// TIA Portal V15.1 export
// export: Created 2024-05-17T05:38:33.441184Z, ExportSetting WithDefaults, DisplayName Totally Integrated Automation Portal, DisplayVersion V15.1 Update 5, DisplayName TIA Portal Openness, DisplayVersion V15.1 Update 5, DisplayName SINAMICS Startdrive Advanced, DisplayVersion V15.1, DisplayName G130, G150, S120, S150, SINAMICS MV, S210, DisplayVersion V15.1, DisplayName G110M, G120, G120C, G120D, G120P, DisplayVersion V15.1, DisplayName STEP 7 Professional, DisplayVersion V15.1 Update 5, DisplayName STEP 7 Safety, DisplayVersion V15.1, DisplayName WinCC Professional, DisplayVersion V15.1 Update 5, DisplayName SIMATIC Visualization Architect, DisplayVersion V15.1
FUNCTION_BLOCK "LProcMasterSlave"   // FB1706, FBD
TITLE = LProcMasterSlave
{ S7_Optimized_Access := 'FALSE' }
AUTHOR : VCC
FAMILY : Control
NAME : MSCtrl
VERSION : 0.1
// ================================================================================
// Master-Slave Controller:
// The temperature is controlled by the Master continuous controller CONT_C and 
// puts out a setpoint value 0-100% to the slave controller CONT_S.
// ================================================================================
// stored: AutoNumber false, IsIECCheckEnabled false, SetENOAutomatically False, UDAEnableTagReadback false
   VAR_INPUT
      I_CYCLE { ExternalAccessible := 'False'; ExternalVisible := 'False'; ExternalWritable := 'False'} : Time;   // Sample time
      I_M_SP_Manual { ExternalAccessible := 'False'; ExternalVisible := 'False'; ExternalWritable := 'False'} : Real;   // Master: Setpoint Manual
      I_M_SP_Auto { ExternalAccessible := 'False'; ExternalVisible := 'False'; ExternalWritable := 'False'} : Real;   // Master: Setpoint for controller
      I_M_PV { ExternalAccessible := 'False'; ExternalVisible := 'False'; ExternalWritable := 'False'} : Real;   // Master: Process value
      I_M_GAIN { ExternalAccessible := 'False'; ExternalVisible := 'False'; ExternalWritable := 'False'} : Real;   // Master: Proportional Gain
      I_M_TI { ExternalAccessible := 'False'; ExternalVisible := 'False'; ExternalWritable := 'False'} : Time;   // Master: Reset time
      I_M_TD { ExternalAccessible := 'False'; ExternalVisible := 'False'; ExternalWritable := 'False'} : Time;   // Master: Derivative time
      I_M_TM_LAG { ExternalAccessible := 'False'; ExternalVisible := 'False'; ExternalWritable := 'False'} : Time;   // Master: Time lag of the derivative action
      I_M_DEADB_W { ExternalAccessible := 'False'; ExternalVisible := 'False'; ExternalWritable := 'False'} : Real;   // Master: Deadband width
      I_M_LMN_HLM { ExternalAccessible := 'False'; ExternalVisible := 'False'; ExternalWritable := 'False'} : Real := 100.0;   // Master: Manipulated value high limit
      I_M_LMN_LLM { ExternalAccessible := 'False'; ExternalVisible := 'False'; ExternalWritable := 'False'} : Real;   // Master: Manipulated value low limit
      I_M_ER_MAX { ExternalAccessible := 'False'; ExternalVisible := 'False'; ExternalWritable := 'False'} : Real := 10.0;   // Master: Maximum deviation for error signal
      I_S_PV { ExternalAccessible := 'False'; ExternalVisible := 'False'; ExternalWritable := 'False'} : Real;   // Slave: Process value
      I_S_GAIN { ExternalAccessible := 'False'; ExternalVisible := 'False'; ExternalWritable := 'False'} : Real;   // Slave: Proportional Gain
      I_S_TI { ExternalAccessible := 'False'; ExternalVisible := 'False'; ExternalWritable := 'False'} : Time;   // Slave: Reset time
      I_S_DEADB_W { ExternalAccessible := 'False'; ExternalVisible := 'False'; ExternalWritable := 'False'} : Real;   // Slave: Deadband width
      I_S_ER_MAX { ExternalAccessible := 'False'; ExternalVisible := 'False'; ExternalWritable := 'False'} : Real := 10.0;   // Slave: Maximum deviation for error signal
      I_S_PULSE_TM { ExternalAccessible := 'False'; ExternalVisible := 'False'; ExternalWritable := 'False'} : Time;   // Slave: Minimum Pulse Time
      I_S_BREAK_TM { ExternalAccessible := 'False'; ExternalVisible := 'False'; ExternalWritable := 'False'} : Time;   // Slave: Minimum Break Time
      I_S_MTR_TM { ExternalAccessible := 'False'; ExternalVisible := 'False'; ExternalWritable := 'False'} : Time;   // Slave: Motor manipulated value
      I_COM_RST { ExternalAccessible := 'False'; ExternalVisible := 'False'; ExternalWritable := 'False'} : Bool;   // Initialising reset of controller
      I_M_MAN_ON { ExternalAccessible := 'False'; ExternalVisible := 'False'; ExternalWritable := 'False'} : Bool;   // Master: Manual value on
      I_M_P_SEL { ExternalAccessible := 'False'; ExternalVisible := 'False'; ExternalWritable := 'False'} : Bool;   // Master: P selected
      I_M_I_SEL { ExternalAccessible := 'False'; ExternalVisible := 'False'; ExternalWritable := 'False'} : Bool;   // Master: I selected
      I_M_D_SEL { ExternalAccessible := 'False'; ExternalVisible := 'False'; ExternalWritable := 'False'} : Bool;   // Master: D selected
      I_S_LMNR_HS { ExternalAccessible := 'False'; ExternalVisible := 'False'; ExternalWritable := 'False'} : Bool;   // Slave: Digital feedback MAX, I/O
      I_S_LMNR_LS { ExternalAccessible := 'False'; ExternalVisible := 'False'; ExternalWritable := 'False'} : Bool;   // Slave: Digital feedback MIN, I/O
      I_S_LMNUP { ExternalAccessible := 'False'; ExternalVisible := 'False'; ExternalWritable := 'False'} : Bool;   // Slave: Manipulated signal up
      I_S_LMNDN { ExternalAccessible := 'False'; ExternalVisible := 'False'; ExternalWritable := 'False'} : Bool;   // Slave: Manipulated signal down
   END_VAR
   VAR_OUTPUT
      O_M_ER { ExternalAccessible := 'False'; ExternalVisible := 'False'; ExternalWritable := 'False'} : Real;   // Deviation Master Controller
      O_SP { ExternalAccessible := 'False'; ExternalVisible := 'False'; ExternalWritable := 'False'} : Real;   // Setpoint used in controller
      O_QLMNUP { ExternalAccessible := 'False'; ExternalVisible := 'False'; ExternalWritable := 'False'} : Bool;   // Output Open
      O_QLMNDN { ExternalAccessible := 'False'; ExternalVisible := 'False'; ExternalWritable := 'False'} : Bool;   // Output Close
      O_M_ER_Alarm { ExternalAccessible := 'False'; ExternalVisible := 'False'; ExternalWritable := 'False'} : Bool;   // Master alarm for deviation
      O_S_ER_Alarm { ExternalAccessible := 'False'; ExternalVisible := 'False'; ExternalWritable := 'False'} : Bool;   // Slave alarm for deviation
   END_VAR
   VAR DB_SPECIFIC
      M_ManValue { ExternalAccessible := 'False'; ExternalVisible := 'False'; ExternalWritable := 'False'} : Real;   // Master: Manual value
      M_LMN { ExternalAccessible := 'False'; ExternalVisible := 'False'; ExternalWritable := 'False'} : Real;   // Master: Manipulated value from controller
      M_PV { ExternalAccessible := 'False'; ExternalVisible := 'False'; ExternalWritable := 'False'} : Real;   // Master: Process variable from controller
      M_ER { ExternalAccessible := 'False'; ExternalVisible := 'False'; ExternalWritable := 'False'} : Real;   // Master: Error signal from controller
      M_ER_ABS { ExternalAccessible := 'False'; ExternalVisible := 'False'; ExternalWritable := 'False'} : Real;   // Master: Absolute error from controller
      S_PV { ExternalAccessible := 'False'; ExternalVisible := 'False'; ExternalWritable := 'False'} : Real;   // Slave: Process variable from controller
      S_ER { ExternalAccessible := 'False'; ExternalVisible := 'False'; ExternalWritable := 'False'} : Real;   // Slave: Error signal from controller
      S_ER_ABS { ExternalAccessible := 'False'; ExternalVisible := 'False'; ExternalWritable := 'False'} : Real;   // Slave: Absolute error from controller
      QLMNUP { ExternalAccessible := 'False'; ExternalVisible := 'False'; ExternalWritable := 'False'} : Bool;   // Step controller output Open
      QLMNDN { ExternalAccessible := 'False'; ExternalVisible := 'False'; ExternalWritable := 'False'} : Bool;   // Step controller output Close
   END_VAR
   VAR
      Continuous_Control { ExternalAccessible := 'False'; ExternalVisible := 'False'; ExternalWritable := 'False'; S7_SetPoint := 'True'} : CONT_C;   // Continuous controller
      Step_Control { ExternalAccessible := 'False'; ExternalVisible := 'False'; ExternalWritable := 'False'; S7_SetPoint := 'True'} : CONT_S;   // Step controller
   END_VAR
   VAR_TEMP   // added for the SCL form of the ladder/FBD networks
      _w1 : Bool;
   END_VAR
BEGIN

REGION Network 1: **** 2.2 - Alarms - Alarms Generation **** Master controller: Calculation absolute error
   // Master controller: Calculation absolute error
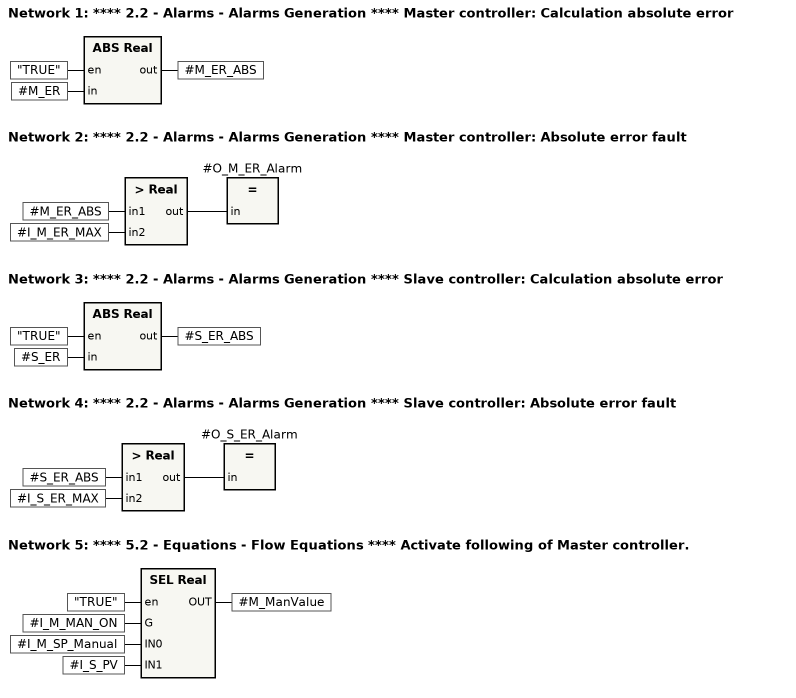
   IF "TRUE" THEN #M_ER_ABS := ABS(#M_ER); END_IF;
END_REGION

REGION Network 2: **** 2.2 - Alarms - Alarms Generation **** Master controller: Absolute error fault
   // Master controller: Absolute error fault
   #O_M_ER_Alarm := #M_ER_ABS > #I_M_ER_MAX;
END_REGION

REGION Network 3: **** 2.2 - Alarms - Alarms Generation **** Slave controller: Calculation absolute error
   // Slave controller: Calculation absolute error
   IF "TRUE" THEN #S_ER_ABS := ABS(#S_ER); END_IF;
END_REGION

REGION Network 4: **** 2.2 - Alarms - Alarms Generation **** Slave controller: Absolute error fault
   // Slave controller: Absolute error fault
   #O_S_ER_Alarm := #S_ER_ABS > #I_S_ER_MAX;
END_REGION

REGION Network 5: **** 5.2 - Equations - Flow Equations **** Activate following of Master controller.
   // Activate following of Master controller.
   IF "TRUE" THEN #M_ManValue := SEL(G := #I_M_MAN_ON, IN0 := #I_M_SP_Manual, IN1 := #I_S_PV); END_IF;
END_REGION

REGION Network 6: **** 7 - Submodules - Non-machine **** Master-Slave control
   // Master-Slave control
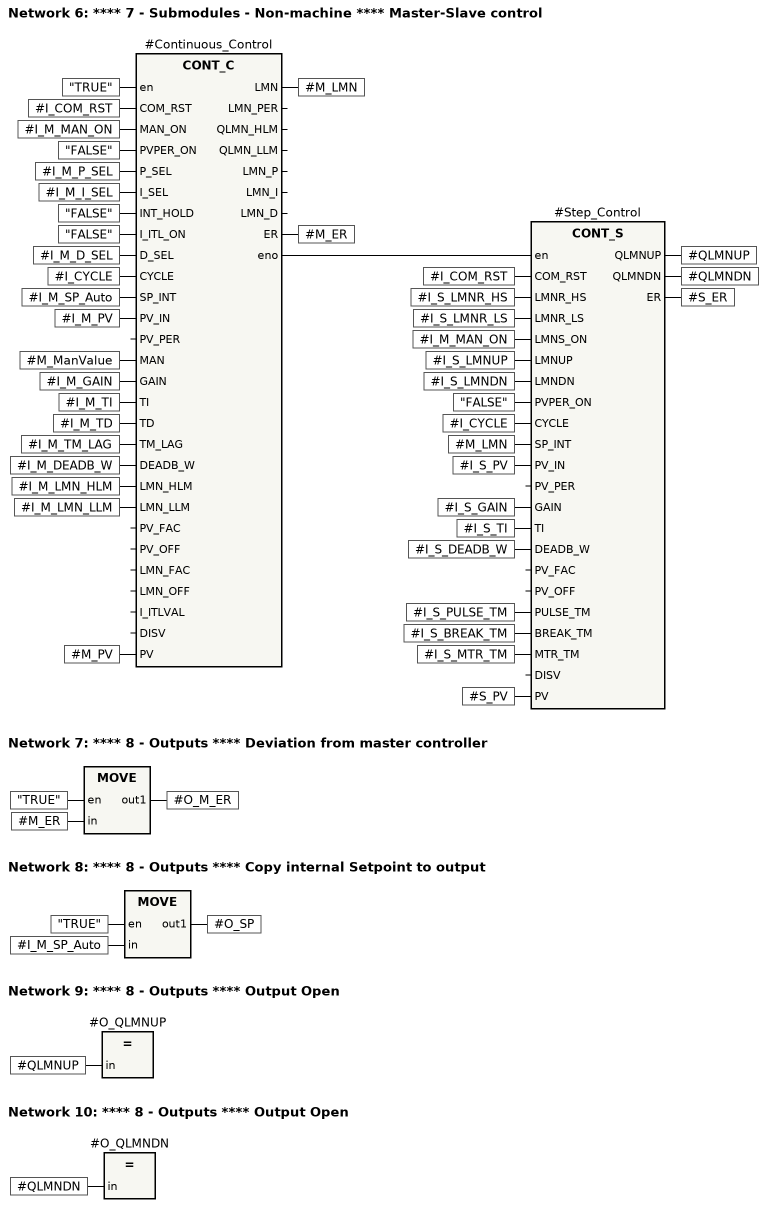
   #Continuous_Control(EN := "TRUE",   // CONT_C
                       COM_RST := #I_COM_RST,
                       MAN_ON := #I_M_MAN_ON,
                       PVPER_ON := "FALSE",
                       P_SEL := #I_M_P_SEL,
                       I_SEL := #I_M_I_SEL,
                       INT_HOLD := "FALSE",
                       I_ITL_ON := "FALSE",
                       D_SEL := #I_M_D_SEL,
                       CYCLE := #I_CYCLE,
                       SP_INT := #I_M_SP_Auto,
                       PV_IN := #I_M_PV,
                       MAN := #M_ManValue,
                       GAIN := #I_M_GAIN,
                       TI := #I_M_TI,
                       TD := #I_M_TD,
                       TM_LAG := #I_M_TM_LAG,
                       DEADB_W := #I_M_DEADB_W,
                       LMN_HLM := #I_M_LMN_HLM,
                       LMN_LLM := #I_M_LMN_LLM,
                       PV := #M_PV,
                       LMN => #M_LMN,
                       ER => #M_ER,
                       ENO => #_w1);
   IF #_w1 THEN
       #Step_Control(COM_RST := #I_COM_RST,   // CONT_S
                     LMNR_HS := #I_S_LMNR_HS,
                     LMNR_LS := #I_S_LMNR_LS,
                     LMNS_ON := #I_M_MAN_ON,
                     LMNUP := #I_S_LMNUP,
                     LMNDN := #I_S_LMNDN,
                     PVPER_ON := "FALSE",
                     CYCLE := #I_CYCLE,
                     SP_INT := #M_LMN,
                     PV_IN := #I_S_PV,
                     GAIN := #I_S_GAIN,
                     TI := #I_S_TI,
                     DEADB_W := #I_S_DEADB_W,
                     PULSE_TM := #I_S_PULSE_TM,
                     BREAK_TM := #I_S_BREAK_TM,
                     MTR_TM := #I_S_MTR_TM,
                     PV := #S_PV,
                     QLMNUP => #QLMNUP,
                     QLMNDN => #QLMNDN,
                     ER => #S_ER);
   END_IF;
END_REGION

REGION Network 7: **** 8 - Outputs **** Deviation from master controller
   // Deviation from master controller
   IF "TRUE" THEN #O_M_ER := #M_ER; END_IF;
END_REGION

REGION Network 8: **** 8 - Outputs **** Copy internal Setpoint to output
   // Copy internal Setpoint to output
   IF "TRUE" THEN #O_SP := #I_M_SP_Auto; END_IF;
END_REGION

REGION Network 9: **** 8 - Outputs **** Output Open
   // Output Open
   #O_QLMNUP := #QLMNUP;
END_REGION

REGION Network 10: **** 8 - Outputs **** Output Open
   // Output Open
   #O_QLMNDN := #QLMNDN;
END_REGION
END_FUNCTION_BLOCK
